KUKA KRL program: TEST_MOTION.src, TEST_MOTION.dat

--- TEST_MOTION.src ---
&ACCESS RVP
&REL 235
&PARAM TEMPLATE = C:\KRC\Roboter\Template\vorgabe
&PARAM EDITMASK = *
DEF TEST_MOTION( )
INT COUNTER
BOOL STATE
DECL IPO_MODE LAST_IPO

;FOLD INI
  ;FOLD BASISTECH INI
    GLOBAL INTERRUPT DECL 3 WHEN $STOPMESS==TRUE DO IR_STOPM ( )
    INTERRUPT ON 3
    BAS (#INITMOV,0 )
  ;ENDFOLD (BASISTECH INI)
  ;FOLD USER INI
    ;Make your modifications here

  ;ENDFOLD (USER INI)
;ENDFOLD (INI)

; Set the advance run pointer to the maximum value
$ADVANCE = 5

;FOLD PTP HOME  Vel= 100 % DEFAULT;%{PE}%MKUKATPBASIS,%CMOVE,%VPTP,%P 1:PTP, 2:HOME, 3:, 5:100, 7:DEFAULT
$BWDSTART = FALSE
PDAT_ACT=PDEFAULT
FDAT_ACT=FHOME
BAS (#PTP_PARAMS,100 )
$H_POS=XHOME
PTP  XHOME
;ENDFOLD

; Note that this program was originally written for
; a demonstration of the search functionality without
; having a real gripper in place.  If a new program is
; written based on this function, note that the tool
; used in this program is a plastic bumper, and that
; all TP-programmed points were based on that tool
; definition.  Modifying Tool[2] in any way will require
; these points to be redefined.
;FOLD PTP P1 Vel=30 % PDAT1 Tool[2]:post Base[0];%{PE}%R 5.6.11,%MKUKATPBASIS,%CMOVE,%VPTP,%P 1:PTP, 2:P1, 3:, 5:30, 7:PDAT1
$BWDSTART=FALSE
PDAT_ACT=PPDAT1
FDAT_ACT=FP1
BAS(#PTP_PARAMS,30)
PTP XP1
;ENDFOLD
;FOLD PTP P2 Vel=100 % PDAT2 Tool[2]:post Base[0];%{PE}%R 5.6.11,%MKUKATPBASIS,%CMOVE,%VPTP,%P 1:PTP, 2:P2, 3:, 5:100, 7:PDAT2
$BWDSTART=FALSE
PDAT_ACT=PPDAT2
FDAT_ACT=FP2
BAS(#PTP_PARAMS,100)
PTP XP2
;ENDFOLD

; Instead of editing Tool[2], just define a new tool
; and set it appropriately here.
$TOOL = TOOL_DATA[3]
$BASE = BASE_DATA[0]

; Switch the coordinate frame to that of the tool
; (the Z axis is that in which the tool flange is
; pointing)
LAST_IPO = $IPO_MODE
$IPO_MODE = #TCP

; Set up Impedance Control
STATE = STARTIMPEDANCE(TRUE)
;$STIFFNESS = NEWSTIFF

; JAM: what am I doing here?
$VEL.cp = 0.2

; Clear all search parameters
STATE = CANCEL_SEARCH()

; Functional tests.  Each test should be assigned
; a value (passed, failed, pending) depending on
; where it is in the evaluation queue.
; =================================================
; INDIVIDUAL SEARCH TESTS
; =================================================
; Spiral Test:  Passed
;BOOL ADDSEARCHSPIRAL(INT TURNS, REAL RADIUS, REAL SPEED)
STATE = STATE AND ADDSEARCHSPIRAL(5, 20.0, 180.0)

; Raster Test:  Passed
;BOOL ADDSEARCHRASTER(REAL RASTERS, REAL LENGTH, REAL WIDTH, REAL SPEED)
;STATE = STATE AND ADDSEARCHRASTER(6, 50.0, 50.0, 100.0)

; Rotate Test:  Passed
;BOOL ADDSEARCHROTATION(REAL RANGE, REAL SPEED)
;STATE = STATE AND ADDSEARCHROTATION(20.0, 40.0)

; Circle Test:  Passed
;BOOL ADDSEARCHCIRCLE(REAL RADIUS, REAL SPEED)
;STATE = STATE AND ADDSEARCHCIRCLE(25.0, 20.0)

; Hop Test   :  Passed
;BOOL ADDSEARCHHOP(REAL MAGNITUDE, REAL FREQUENCY)
;STATE = STATE AND ADDSEARCHHOP(20.0, 5.0)

; Linear Test:  Passed
;BOOL ADDSEARCHLINEAR(REAL X_OFFSET, REAL Y_OFFSET, REAL Z_OFFSET, REAL SPEED)
;STATE = STATE AND ADDSEARCHLINEAR(0.0, 0.0, -100.0, 10.0)

; Constant Offset Test:  PASSED
;BOOL ADDSEARCHCONSTOFFSET(REAL X_OFFSET, REAL Y_OFFSET, REAL Z_OFFSET)
;STATE = STATE AND ADDSEARCHCONSTOFFSET(0.0, 0.0, -50.0)

; =================================================
; COMBINATORIAL SEARCH TEST
; =================================================
; Linear + Rotation Test:  Passed
;STATE = STATE AND ADDSEARCHLINEAR(50.0, -10.0, 20.0, 2.0)
;STATE = STATE AND ADDSEARCHROTATION(20.0, 100.0)

; =================================================
; TERMINATION CONDITION TESTS
; =================================================
; Alarm clock test:  Passed
STATE = STATE AND ADDTERMCLOCK(#ALARMCLOCK, #FAIL, 10000.0, 5)

; Program timer test:  Passed
;STATE = STATE AND ADDTERMCLOCK(#PROGTIME, #FAIL, 20000.0, 5)

; Distance test:  Pending
STATE = STATE AND ADDTERMDISTANCE(#SUCCESS, 0.0, 0.0, 80.0, 0.0)

; Digital input test:  Pending
;STATE = STATE AND ADDTERMSIGNAL(#EXTSIGNAL, #SUCCESS, 5)

; Contact threshold test:  Pending
;STATE = STATE AND ADDTERMSIGNAL(#CONTACT, #SUCCESS, 2.0)

; ==========================================
; ~~~    RUN DAT SWEET, SWEET SEARCH     ~~~
; ==========================================
WHILE STATE
  STATE = (SEARCH() == #RUNNING)
ENDWHILE
; ==========================================

; Go back to position control and clear all search
; parameters
STATE = STARTIMPEDANCE(FALSE)
STATE = CANCEL_SEARCH()

; Back out of the insertion point in position control
targetpos = $POS_ACT_MES
targetpos.z = targetpos.z + 100.0
PTP targetpos

; Switch back to the original coordinate frame
$IPO_MODE = LAST_IPO

;FOLD PTP HOME Vel=30 % DEFAULT;%{PE}%R 5.6.11,%MKUKATPBASIS,%CMOVE,%VPTP,%P 1:PTP, 2:HOME, 3:, 5:30, 7:DEFAULT
$BWDSTART=FALSE
PDAT_ACT=PDEFAULT
FDAT_ACT=FHOME
BAS(#PTP_PARAMS,30)
$H_POS=XHOME
PTP XHOME
;ENDFOLD

END

--- TEST_MOTION.dat ---
&ACCESS RVP
&REL 235
&PARAM TEMPLATE = C:\KRC\Roboter\Template\vorgabe
&PARAM EDITMASK = *
DEFDAT  TEST_MOTION
;FOLD EXTERNAL DECLARATIONS;%{PE}%MKUKATPBASIS,%CEXT,%VCOMMON,%P
;FOLD BASISTECH EXT;%{PE}%MKUKATPBASIS,%CEXT,%VEXT,%P
EXT  BAS (BAS_COMMAND  :IN,REAL  :IN )
DECL INT SUCCESS
;ENDFOLD (BASISTECH EXT)
;FOLD USER EXT;%{E}%MKUKATPUSER,%CEXT,%VEXT,%P
;Make here your modifications

;ENDFOLD (USER EXT)
;ENDFOLD (EXTERNAL DECLARATIONS)
DECL BASIS_SUGG_T LAST_BASIS={POINT1[] "P2                      ",POINT2[] "P2                      ",CP_PARAMS[] "CPDAT0                  ",PTP_PARAMS[] "PDAT2                   ",CONT[] "                        ",CP_VEL[] "2.0                     ",PTP_VEL[] "100                     ",SYNC_PARAMS[] "SYNCDAT                 ",SPL_NAME[] "S0                      "}
DECL E6POS XP1={X 342.598389,Y -458.466797,Z 289.5914,A 148.138306,B -1.71656001,C -179.952499,S 6,T 49,E1 -68.91539,E2 0.0,E3 0.0,E4 0.0,E5 0.0,E6 0.0}
DECL FDAT FP1={TOOL_NO 2,BASE_NO 0,IPO_FRAME #BASE,POINT2[] " ",TQ_STATE FALSE}
DECL PDAT PPDAT1={VEL 100.0,ACC 100.0,APO_DIST 100.0,APO_MODE #CPTP}

DECL INT md_int[16]
DECL REAL md_real[16]
DECL INT result
DECL INT ii
DECL E6POS XP2={X 518.148682,Y -483.22879,Z 475.679596,A 78.9688797,B 39.79496,C 84.3012466,S 6,T 49,E1 -68.9144363,E2 0.0,E3 0.0,E4 0.0,E5 0.0,E6 0.0}
DECL FDAT FP2={TOOL_NO 2,BASE_NO 0,IPO_FRAME #BASE,POINT2[] " ",TQ_STATE FALSE}
DECL PDAT PPDAT2={VEL 100.0,ACC 100.0,APO_DIST 100.0,APO_MODE #CPTP}
ENDDAT
